Fanuc KAREL source: kt00072.KL

-- PROVISIONAL review KL for V940-1; original PC SHA256 9fd98520978824963e481b2ccf8be8526a986c2aa242f070ffe858e58313096f
-- Incomplete behavior may be omitted. Consult companion uncertainty JSON. Do not deploy.
PROGRAM KT00072
%NOLOCKGROUP
VAR
  I1 : INTEGER
  OUT : REAL
-- UNRESOLVED_DECL H2 type=002017
BEGIN
  -- V9_ZERO_TABLE_METADATA_HINT layout=0001; no indexed target words; source/name/runtime held
  -- UNRESOLVED_PC offsets 5-16; opcodes 2E,23
  -- UNRESOLVED_PC offsets 21-35; opcodes 2E,22,9D,33,B4
  -- UNRESOLVED_PC offsets 40-63; opcodes 21,22,9D,33,B3,54,64,23
  -- UNRESOLVED_PC offsets 68-72; opcodes 7F
END KT00072
